FUNCTION_BLOCK FB_LichtBewegungsmelder
VAR_INPUT
	bEinKurz				: BOOL;
	bEinLang				: BOOL;
	bAus 						: BOOL;
	tKurz						: TIME := t#5m;
	tLang 					: TIME := t#60m;
END_VAR
VAR_OUTPUT
END_VAR
VAR_IN_OUT
	bGruppeAus : BOOL;
 	IOstTimeSwitchTimes : ST_TimeSwitchTimes;
END_VAR
VAR
	bInit 			: BOOL := TRUE;
	bInVisu			: BOOL;
	bIn					: BOOL;

	bKlickEnable	: BOOL;
	bLangEnable		: BOOL;

	(* %I / %Q ********************)
	IbInTaster		AT %I* : BOOL;
	IbInBewegunsm AT %I* : BOOL;
	QbOutLicht		AT %Q* : BOOL;

	tofEin			: TOF;

	fbTaster 		: FB_Taster;
  fbTimeSwitch : FB_TimeSwitch;
  
END_VAR

IF bInit THEN
	bKlickEnable := (tkurz <> t#0s);
	bLangEnable := (tLang <> t#0s);
	bInit := FALSE;
END_IF

fbTimeSwitch(IOstTimeSwitchTimes := IOstTimeSwitchTimes);

bIn := IbInTaster OR bInVisu;
fbTaster(bIn:= bIn);

IF IbInBewegunsm THEN
  IF fbTimeSwitch.OUTbOn THEN
    IF bKlickEnable THEN
      tofEin(IN:= TRUE, PT:= tLang);
  	END_IF
  ELSE
    IF bKlickEnable THEN
      tofEin(IN:= TRUE, PT:= tkurz);
  	END_IF
	END_IF

ELSIF bKlickEnable
AND (fbTaster.bKlick
		OR bEinKurz
		OR gbLichtZentralEin)
THEN
	tofEin(IN:= TRUE, PT:= tkurz);
ELSIF bLangEnable
AND (fbTaster.bLang
		OR bEinLang)
THEN
	tofEin(IN:= TRUE, PT:= tLang);
END_IF
tofEin(IN:= FALSE);

IF fbTaster.bLang
AND bKlickEnable
AND bLangEnable
OR bEinKurz
OR bEinLang
OR gbLichtZentralEin
OR IbInBewegunsm
THEN
	QbOutLicht := TRUE;
END_IF

IF (fbTaster.bKlick
		AND bKlickEnable)
OR (fbTaster.bLang
		AND NOT bKlickEnable
		AND bLangEnable)
THEN
	QbOutLicht := NOT QbOutLicht;
END_IF

IF QbOutLicht AND NOT tofEin.Q
OR gbLichtZentralAus OR bAus THEN
	QbOutLicht := FALSE;
END_IF

IF fbTaster.bKlick2 THEN
	bGruppeAus := TRUE;
END_IF

END_FUNCTION_BLOCK

(* stored: Version 1.1.0.1, ProductVersion 3.1.4018.9
   POU FB_LichtBewegungsmelder: Id {8a6a4d2b-4d98-4810-bd15-0ff6e5ef346d}, SpecialFunc None *)
